TYPE JSON_DOCUMENT : STRING(25000); END_TYPE

(* stored: Version 1.1.0.1
   DUT JSON_DOCUMENT: Id {4e32bf14-1ec8-4089-85d1-43fdf25ac303} *)
